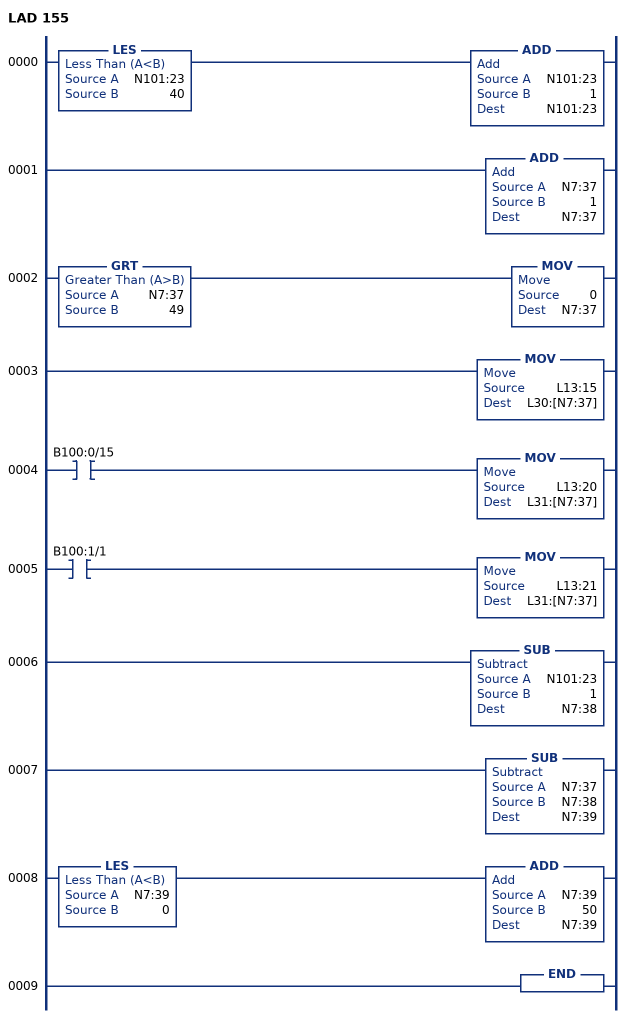
% Rung: 0 %
SOR LES N101:23 40 ADD N101:23 1 N101:23 EOR
% Rung: 1 %
SOR ADD N7:37 1 N7:37 EOR
% Rung: 2 %
SOR GRT N7:37 49 MOV 0 N7:37 EOR
% Rung: 3 %
SOR MOV L13:15 L30:[N7:37] EOR
% Rung: 4 %
SOR XIC B100:0/15 MOV L13:20 L31:[N7:37] EOR
% Rung: 5 %
SOR XIC B100:1/1 MOV L13:21 L31:[N7:37] EOR
% Rung: 6 %
SOR SUB N101:23 1 N7:38 EOR
% Rung: 7 %
SOR SUB N7:37 N7:38 N7:39 EOR
% Rung: 8 %
SOR LES N7:39 0 ADD N7:39 50 N7:39 EOR
% Rung: 9 %
SOR END EOR

LADDER 156
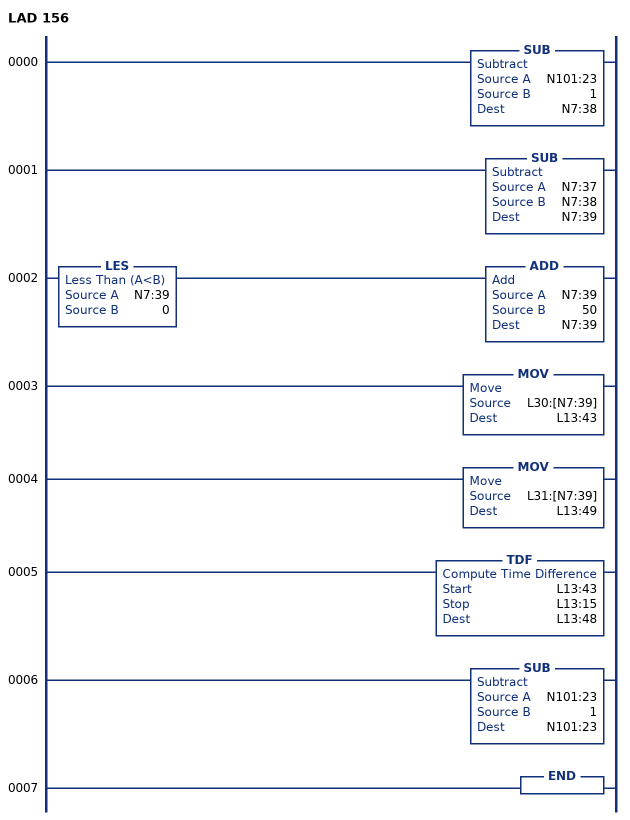
% Rung: 0 %
SOR SUB N101:23 1 N7:38 EOR
% Rung: 1 %
SOR SUB N7:37 N7:38 N7:39 EOR
% Rung: 2 %
SOR LES N7:39 0 ADD N7:39 50 N7:39 EOR
% Rung: 3 %
SOR MOV L30:[N7:39] L13:43 EOR
% Rung: 4 %
SOR MOV L31:[N7:39] L13:49 EOR
% Rung: 5 %
SOR TDF L13:43 L13:15 L13:48 EOR
% Rung: 6 %
SOR SUB N101:23 1 N101:23 EOR
% Rung: 7 %
SOR END EOR

LADDER 157
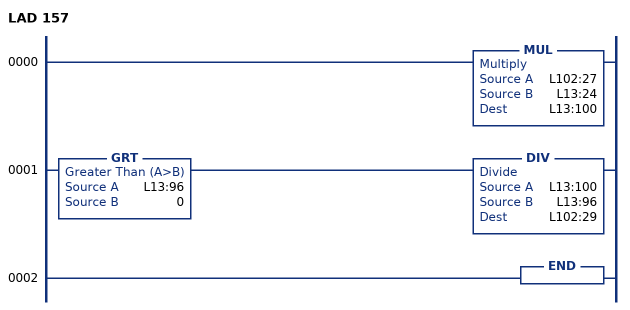
% Rung: 0 %
SOR MUL L102:27 L13:24 L13:100 EOR
% Rung: 1 %
SOR GRT L13:96 0 DIV L13:100 L13:96 L102:29 EOR
% Rung: 2 %
SOR END EOR

LADDER 158
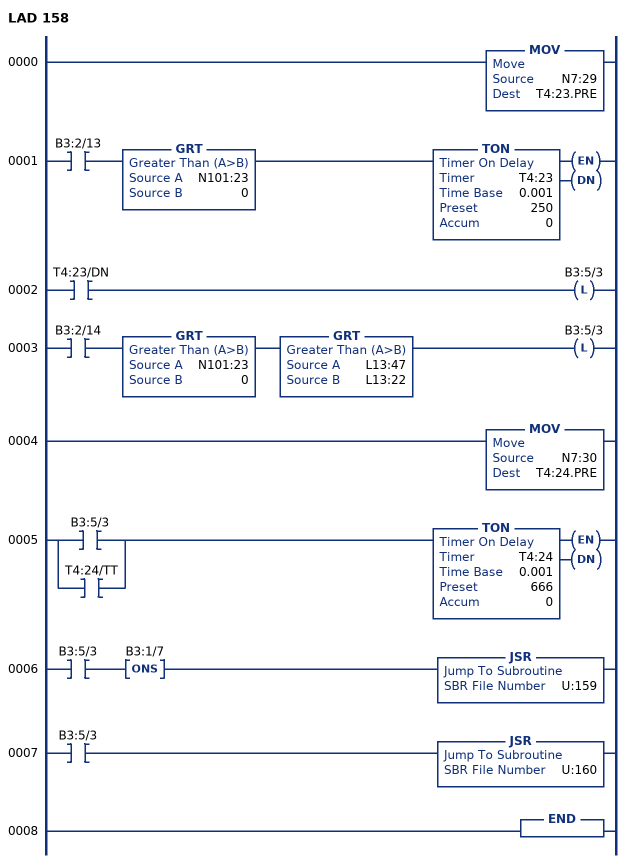
% Rung: 0 %
SOR MOV N7:29 T4:23.PRE EOR
% Rung: 1 %
SOR XIC B3:2/13 GRT N101:23 0 TON T4:23 0.001 250 0 EOR
% Rung: 2 %
SOR XIC T4:23/DN OTL B3:5/3 EOR
% Rung: 3 %
SOR XIC B3:2/14 GRT N101:23 0 GRT L13:47 L13:22 OTL B3:5/3 EOR
% Rung: 4 %
SOR MOV N7:30 T4:24.PRE EOR
% Rung: 5 %
SOR BST XIC B3:5/3 NXB XIC T4:24/TT BND TON T4:24 0.001 666 0 EOR
% Rung: 6 %
SOR XIC B3:5/3 ONS B3:1/7 JSR U:159 EOR
% Rung: 7 %
SOR XIC B3:5/3 JSR U:160 EOR
% Rung: 8 %
SOR END EOR

LADDER 159
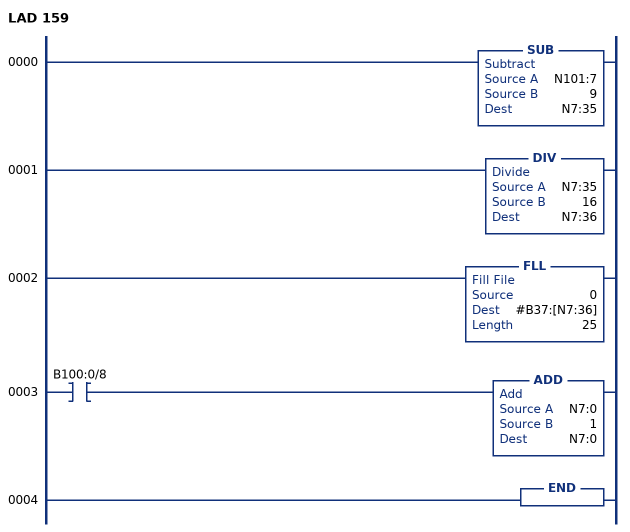
% Rung: 0 %
SOR SUB N101:7 9 N7:35 EOR
% Rung: 1 %
SOR DIV N7:35 16 N7:36 EOR
% Rung: 2 %
SOR FLL 0 #B37:[N7:36] 25 EOR
% Rung: 3 %
SOR XIC B100:0/8 ADD N7:0 1 N7:0 EOR
% Rung: 4 %
SOR END EOR

LADDER 160
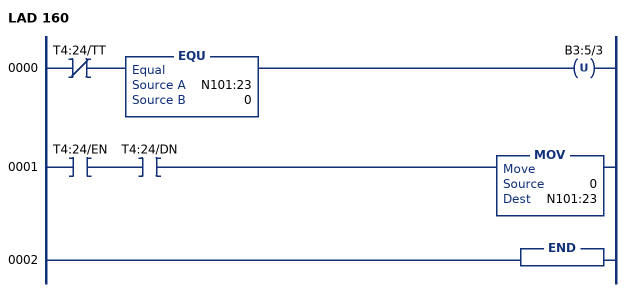
% Rung: 0 %
SOR XIO T4:24/TT EQU N101:23 0 OTU B3:5/3 EOR
% Rung: 1 %
SOR XIC T4:24/EN XIC T4:24/DN MOV 0 N101:23 EOR
% Rung: 2 %
SOR END EOR

LADDER 161
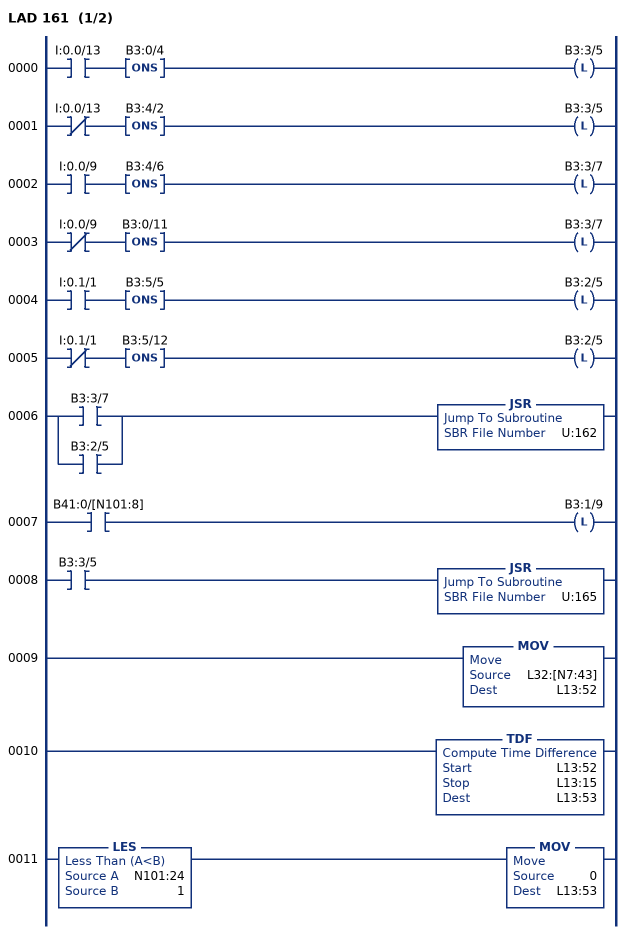
% Rung: 0 %
SOR XIC I:0.0/13 ONS B3:0/4 OTL B3:3/5 EOR
% Rung: 1 %
SOR XIO I:0.0/13 ONS B3:4/2 OTL B3:3/5 EOR
% Rung: 2 %
SOR XIC I:0.0/9 ONS B3:4/6 OTL B3:3/7 EOR
% Rung: 3 %
SOR XIO I:0.0/9 ONS B3:0/11 OTL B3:3/7 EOR
% Rung: 4 %
SOR XIC I:0.1/1 ONS B3:5/5 OTL B3:2/5 EOR
% Rung: 5 %
SOR XIO I:0.1/1 ONS B3:5/12 OTL B3:2/5 EOR
% Rung: 6 %
SOR BST XIC B3:3/7 NXB XIC B3:2/5 BND JSR U:162 EOR
% Rung: 7 %
SOR XIC B41:0/[N101:8] OTL B3:1/9 EOR
% Rung: 8 %
SOR XIC B3:3/5 JSR U:165 EOR
% Rung: 9 %
SOR MOV L32:[N7:43] L13:52 EOR
% Rung: 10 %
SOR TDF L13:52 L13:15 L13:53 EOR
% Rung: 11 %
SOR LES N101:24 1 MOV 0 L13:53 EOR

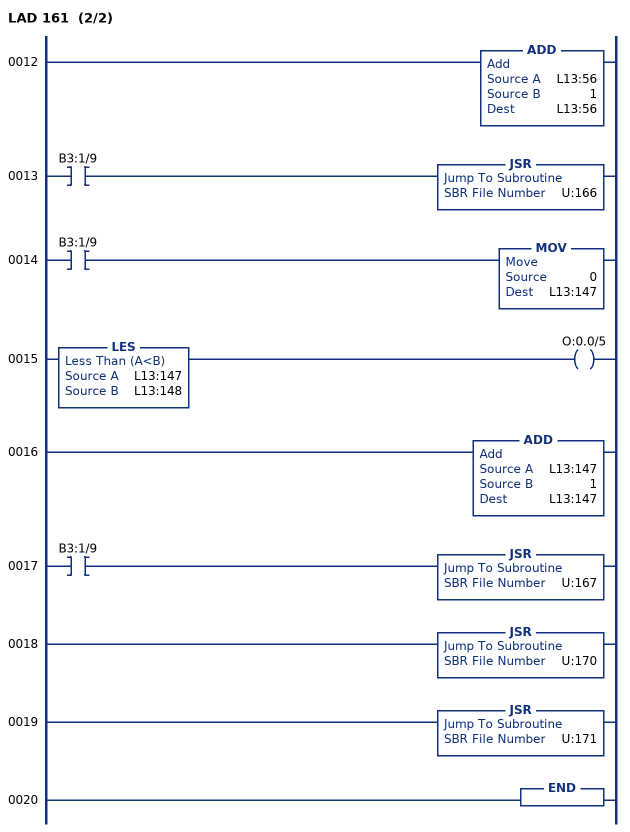
% Rung: 12 %
SOR ADD L13:56 1 L13:56 EOR
% Rung: 13 %
SOR XIC B3:1/9 JSR U:166 EOR
% Rung: 14 %
SOR XIC B3:1/9 MOV 0 L13:147 EOR
% Rung: 15 %
SOR LES L13:147 L13:148 OTE O:0.0/5 EOR
% Rung: 16 %
SOR ADD L13:147 1 L13:147 EOR
% Rung: 17 %
SOR XIC B3:1/9 JSR U:167 EOR
% Rung: 18 %
SOR JSR U:170 EOR
% Rung: 19 %
SOR JSR U:171 EOR
% Rung: 20 %
SOR END EOR

LADDER 162
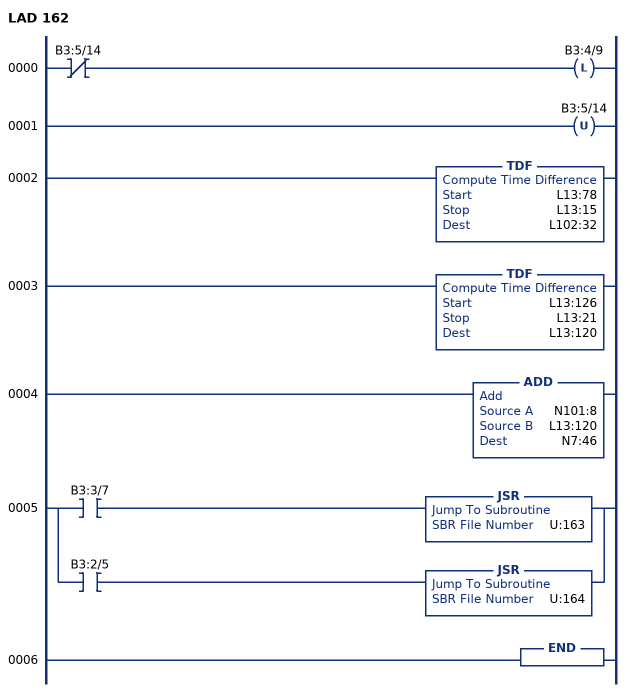
% Rung: 0 %
SOR XIO B3:5/14 OTL B3:4/9 EOR
% Rung: 1 %
SOR OTU B3:5/14 EOR
% Rung: 2 %
SOR TDF L13:78 L13:15 L102:32 EOR
% Rung: 3 %
SOR TDF L13:126 L13:21 L13:120 EOR
% Rung: 4 %
SOR ADD N101:8 L13:120 N7:46 EOR
% Rung: 5 %
SOR BST XIC B3:3/7 JSR U:163 NXB XIC B3:2/5 JSR U:164 BND EOR
% Rung: 6 %
SOR END EOR

LADDER 163
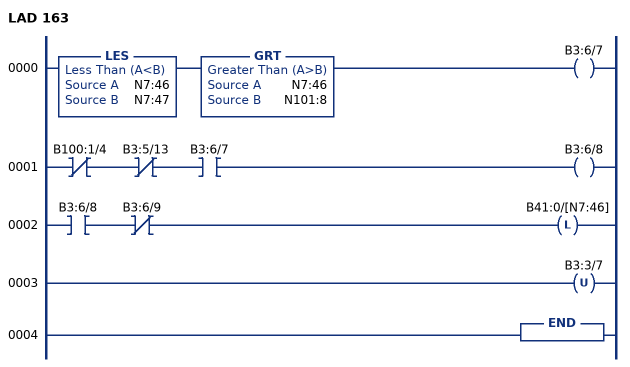
% Rung: 0 %
SOR LES N7:46 N7:47 GRT N7:46 N101:8 OTE B3:6/7 EOR
% Rung: 1 %
SOR XIO B100:1/4 XIO B3:5/13 XIC B3:6/7 OTE B3:6/8 EOR
% Rung: 2 %
SOR XIC B3:6/8 XIO B3:6/9 OTL B41:0/[N7:46] EOR
% Rung: 3 %
SOR OTU B3:3/7 EOR
% Rung: 4 %
SOR END EOR

LADDER 164
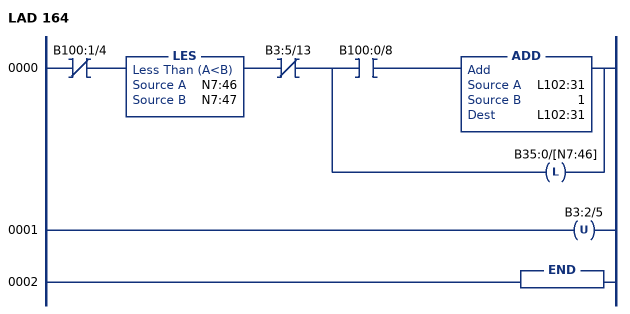
% Rung: 0 %
SOR XIO B100:1/4 LES N7:46 N7:47 XIO B3:5/13 BST XIC B100:0/8 ADD L102:31 1 L102:31 NXB OTL B35:0/[N7:46] BND EOR
% Rung: 1 %
SOR OTU B3:2/5 EOR
% Rung: 2 %
SOR END EOR

LADDER 165
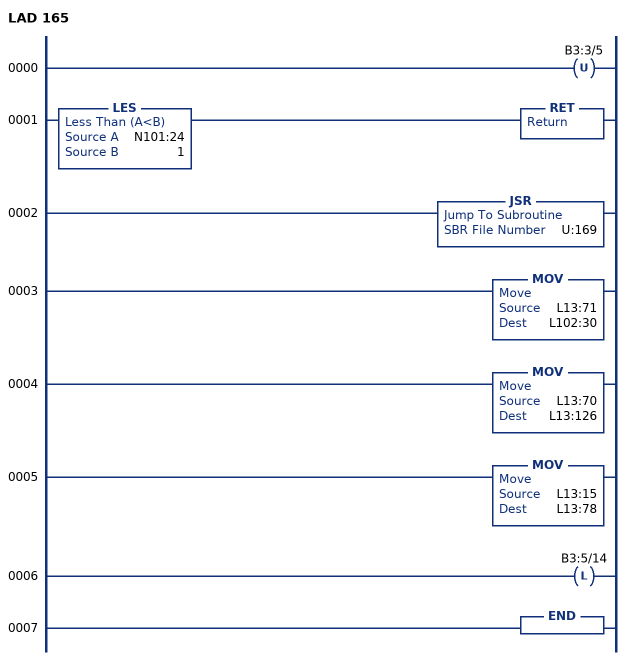
% Rung: 0 %
SOR OTU B3:3/5 EOR
% Rung: 1 %
SOR LES N101:24 1 RET EOR
% Rung: 2 %
SOR JSR U:169 EOR
% Rung: 3 %
SOR MOV L13:71 L102:30 EOR
% Rung: 4 %
SOR MOV L13:70 L13:126 EOR
% Rung: 5 %
SOR MOV L13:15 L13:78 EOR
% Rung: 6 %
SOR OTL B3:5/14 EOR
% Rung: 7 %
SOR END EOR

LADDER 166
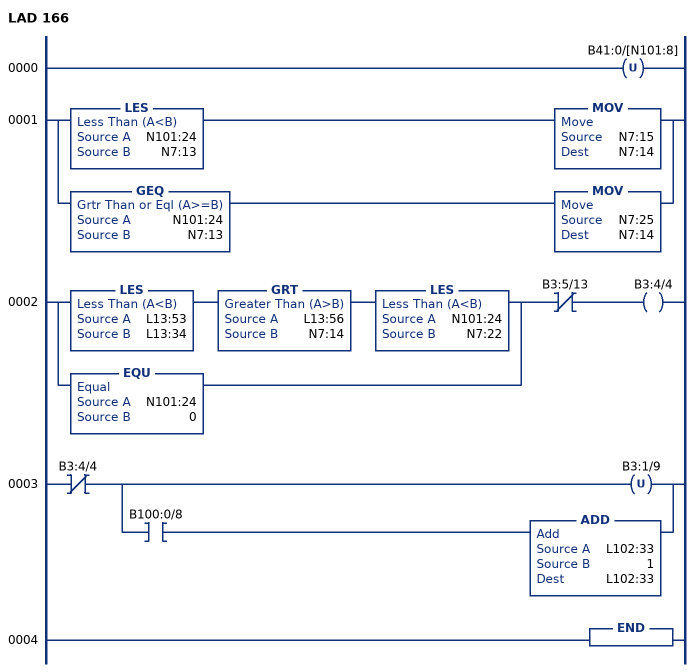
% Rung: 0 %
SOR OTU B41:0/[N101:8] EOR
% Rung: 1 %
SOR BST LES N101:24 N7:13 MOV N7:15 N7:14 NXB GEQ N101:24 N7:13 MOV N7:25 N7:14 BND EOR
% Rung: 2 %
SOR BST LES L13:53 L13:34 GRT L13:56 N7:14 LES N101:24 N7:22 NXB EQU N101:24 0 BND XIO B3:5/13 OTE B3:4/4 EOR
% Rung: 3 %
SOR XIO B3:4/4 BST OTU B3:1/9 NXB XIC B100:0/8 ADD L102:33 1 L102:33 BND EOR
% Rung: 4 %
SOR END EOR

LADDER 167
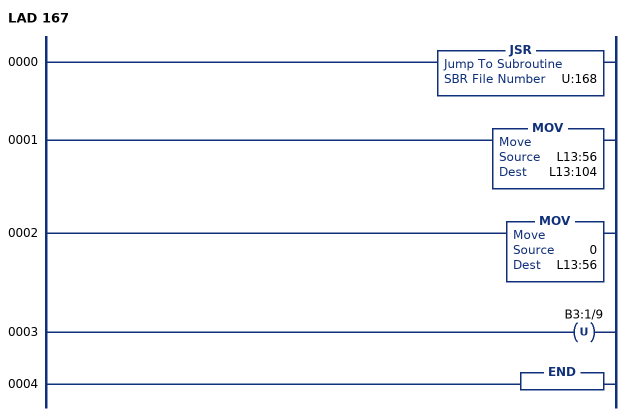
% Rung: 0 %
SOR JSR U:168 EOR
% Rung: 1 %
SOR MOV L13:56 L13:104 EOR
% Rung: 2 %
SOR MOV 0 L13:56 EOR
% Rung: 3 %
SOR OTU B3:1/9 EOR
% Rung: 4 %
SOR END EOR

LADDER 168
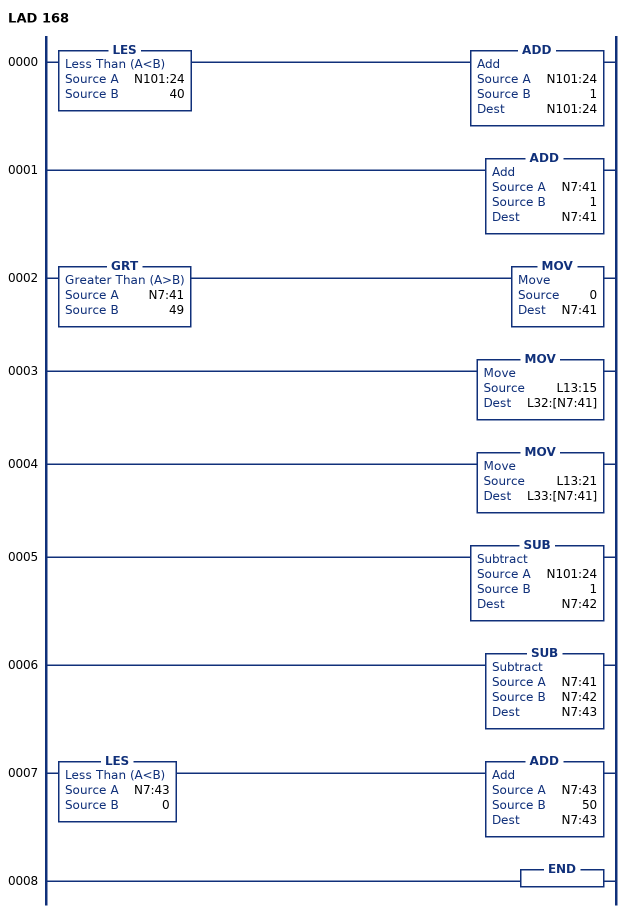
% Rung: 0 %
SOR LES N101:24 40 ADD N101:24 1 N101:24 EOR
% Rung: 1 %
SOR ADD N7:41 1 N7:41 EOR
% Rung: 2 %
SOR GRT N7:41 49 MOV 0 N7:41 EOR
% Rung: 3 %
SOR MOV L13:15 L32:[N7:41] EOR
% Rung: 4 %
SOR MOV L13:21 L33:[N7:41] EOR
% Rung: 5 %
SOR SUB N101:24 1 N7:42 EOR
% Rung: 6 %
SOR SUB N7:41 N7:42 N7:43 EOR
% Rung: 7 %
SOR LES N7:43 0 ADD N7:43 50 N7:43 EOR
% Rung: 8 %
SOR END EOR

LADDER 169
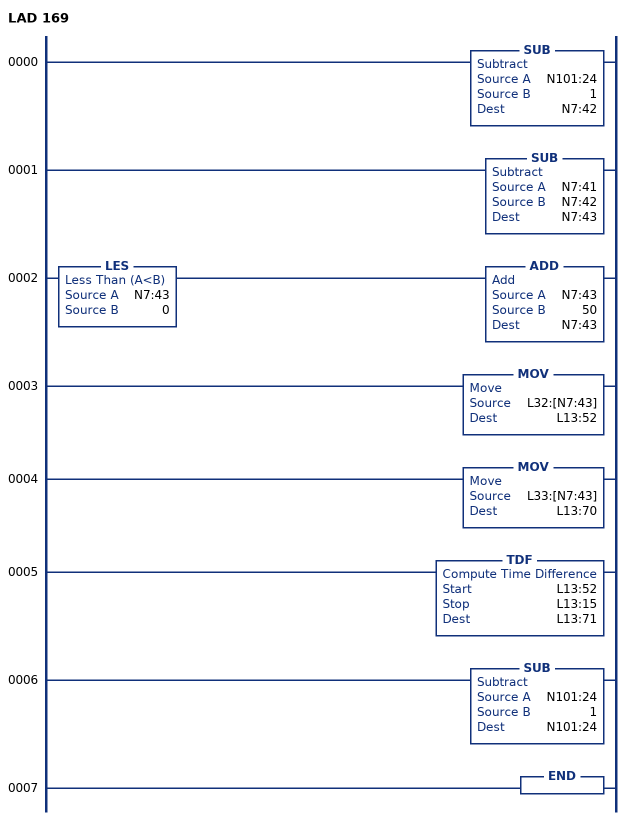
% Rung: 0 %
SOR SUB N101:24 1 N7:42 EOR
% Rung: 1 %
SOR SUB N7:41 N7:42 N7:43 EOR
% Rung: 2 %
SOR LES N7:43 0 ADD N7:43 50 N7:43 EOR
% Rung: 3 %
SOR MOV L32:[N7:43] L13:52 EOR
% Rung: 4 %
SOR MOV L33:[N7:43] L13:70 EOR
% Rung: 5 %
SOR TDF L13:52 L13:15 L13:71 EOR
% Rung: 6 %
SOR SUB N101:24 1 N101:24 EOR
% Rung: 7 %
SOR END EOR

LADDER 170
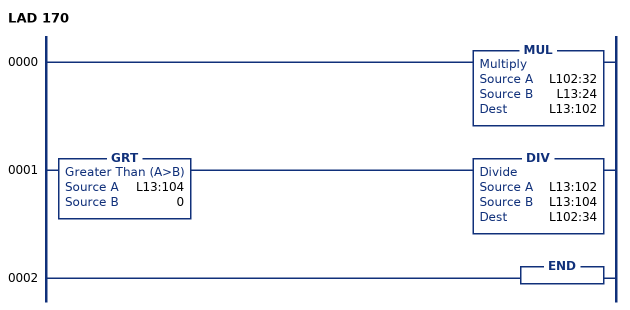
% Rung: 0 %
SOR MUL L102:32 L13:24 L13:102 EOR
% Rung: 1 %
SOR GRT L13:104 0 DIV L13:102 L13:104 L102:34 EOR
% Rung: 2 %
SOR END EOR

LADDER 171
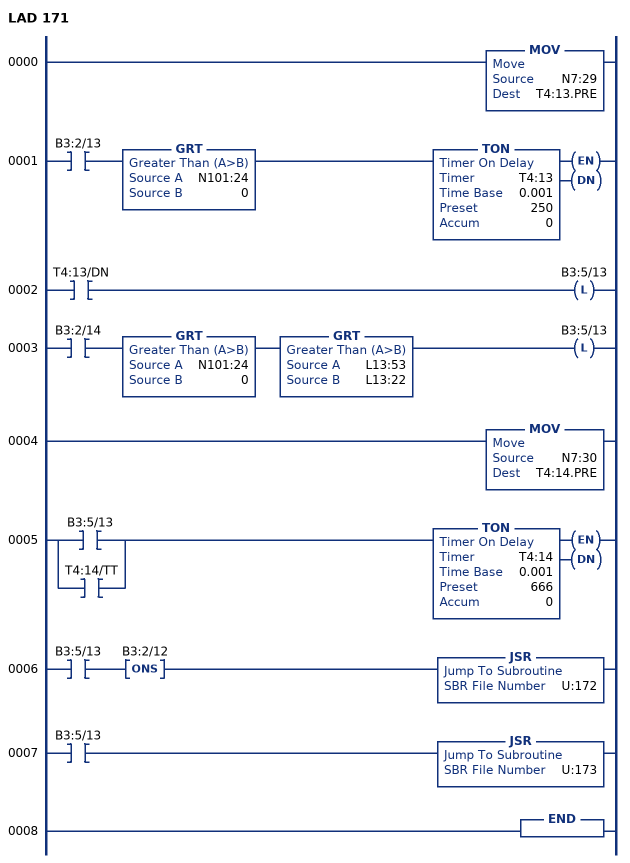
% Rung: 0 %
SOR MOV N7:29 T4:13.PRE EOR
% Rung: 1 %
SOR XIC B3:2/13 GRT N101:24 0 TON T4:13 0.001 250 0 EOR
% Rung: 2 %
SOR XIC T4:13/DN OTL B3:5/13 EOR
% Rung: 3 %
SOR XIC B3:2/14 GRT N101:24 0 GRT L13:53 L13:22 OTL B3:5/13 EOR
% Rung: 4 %
SOR MOV N7:30 T4:14.PRE EOR
% Rung: 5 %
SOR BST XIC B3:5/13 NXB XIC T4:14/TT BND TON T4:14 0.001 666 0 EOR
% Rung: 6 %
SOR XIC B3:5/13 ONS B3:2/12 JSR U:172 EOR
% Rung: 7 %
SOR XIC B3:5/13 JSR U:173 EOR
% Rung: 8 %
SOR END EOR

LADDER 172
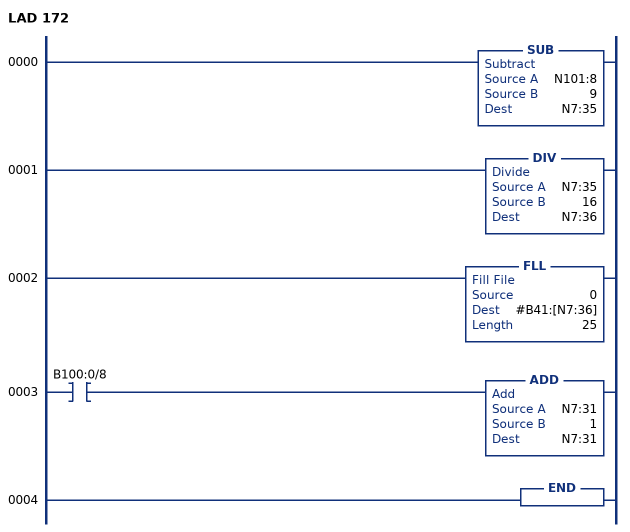
% Rung: 0 %
SOR SUB N101:8 9 N7:35 EOR
% Rung: 1 %
SOR DIV N7:35 16 N7:36 EOR
% Rung: 2 %
SOR FLL 0 #B41:[N7:36] 25 EOR
% Rung: 3 %
SOR XIC B100:0/8 ADD N7:31 1 N7:31 EOR
% Rung: 4 %
SOR END EOR

LADDER 173
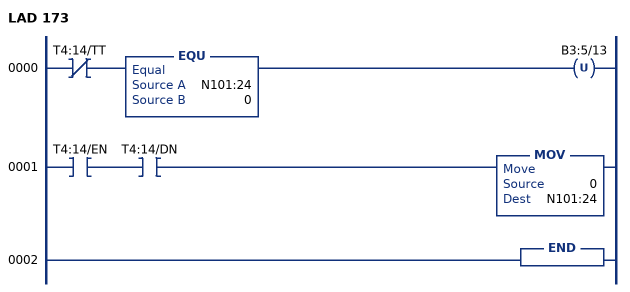
% Rung: 0 %
SOR XIO T4:14/TT EQU N101:24 0 OTU B3:5/13 EOR
% Rung: 1 %
SOR XIC T4:14/EN XIC T4:14/DN MOV 0 N101:24 EOR
% Rung: 2 %
SOR END EOR

LADDER 174
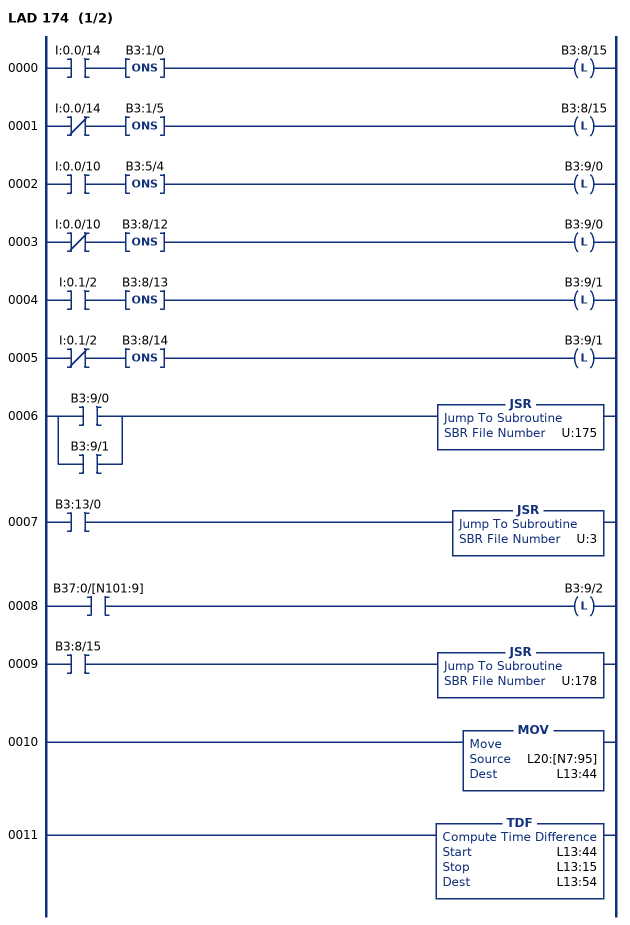
% Rung: 0 %
SOR XIC I:0.0/14 ONS B3:1/0 OTL B3:8/15 EOR
% Rung: 1 %
SOR XIO I:0.0/14 ONS B3:1/5 OTL B3:8/15 EOR
% Rung: 2 %
SOR XIC I:0.0/10 ONS B3:5/4 OTL B3:9/0 EOR
% Rung: 3 %
SOR XIO I:0.0/10 ONS B3:8/12 OTL B3:9/0 EOR
% Rung: 4 %
SOR XIC I:0.1/2 ONS B3:8/13 OTL B3:9/1 EOR
% Rung: 5 %
SOR XIO I:0.1/2 ONS B3:8/14 OTL B3:9/1 EOR
% Rung: 6 %
SOR BST XIC B3:9/0 NXB XIC B3:9/1 BND JSR U:175 EOR
% Rung: 7 %
SOR XIC B3:13/0 JSR U:3 EOR
% Rung: 8 %
SOR XIC B37:0/[N101:9] OTL B3:9/2 EOR
% Rung: 9 %
SOR XIC B3:8/15 JSR U:178 EOR
% Rung: 10 %
SOR MOV L20:[N7:95] L13:44 EOR
% Rung: 11 %
SOR TDF L13:44 L13:15 L13:54 EOR

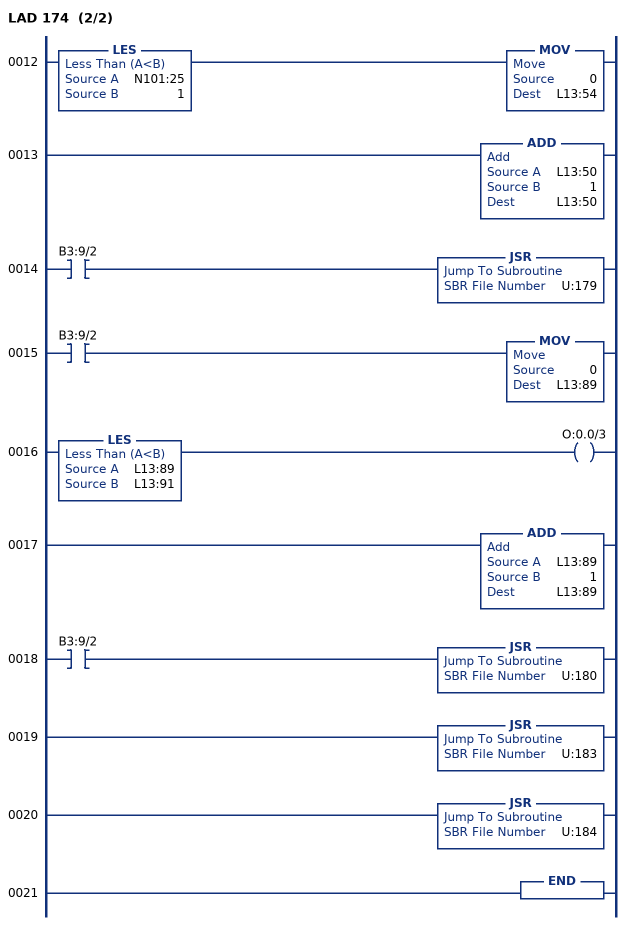
% Rung: 12 %
SOR LES N101:25 1 MOV 0 L13:54 EOR
% Rung: 13 %
SOR ADD L13:50 1 L13:50 EOR
% Rung: 14 %
SOR XIC B3:9/2 JSR U:179 EOR
% Rung: 15 %
SOR XIC B3:9/2 MOV 0 L13:89 EOR
% Rung: 16 %
SOR LES L13:89 L13:91 OTE O:0.0/3 EOR
% Rung: 17 %
SOR ADD L13:89 1 L13:89 EOR
% Rung: 18 %
SOR XIC B3:9/2 JSR U:180 EOR
% Rung: 19 %
SOR JSR U:183 EOR
% Rung: 20 %
SOR JSR U:184 EOR
% Rung: 21 %
SOR END EOR

LADDER 175
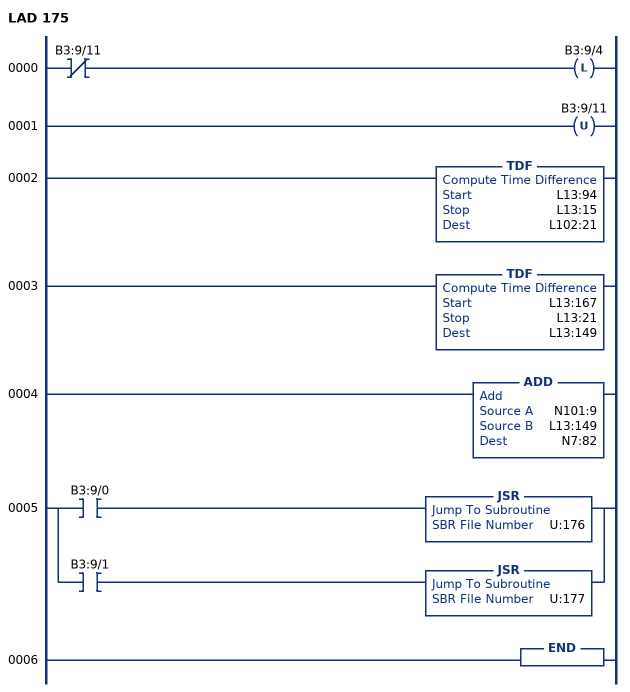
% Rung: 0 %
SOR XIO B3:9/11 OTL B3:9/4 EOR
% Rung: 1 %
SOR OTU B3:9/11 EOR
% Rung: 2 %
SOR TDF L13:94 L13:15 L102:21 EOR
% Rung: 3 %
SOR TDF L13:167 L13:21 L13:149 EOR
% Rung: 4 %
SOR ADD N101:9 L13:149 N7:82 EOR
% Rung: 5 %
SOR BST XIC B3:9/0 JSR U:176 NXB XIC B3:9/1 JSR U:177 BND EOR
% Rung: 6 %
SOR END EOR

LADDER 176
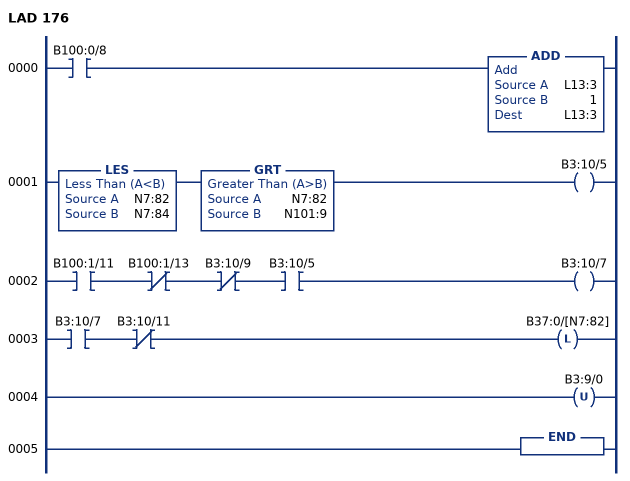
% Rung: 0 %
SOR XIC B100:0/8 ADD L13:3 1 L13:3 EOR
% Rung: 1 %
SOR LES N7:82 N7:84 GRT N7:82 N101:9 OTE B3:10/5 EOR
% Rung: 2 %
SOR XIC B100:1/11 XIO B100:1/13 XIO B3:10/9 XIC B3:10/5 OTE B3:10/7 EOR
% Rung: 3 %
SOR XIC B3:10/7 XIO B3:10/11 OTL B37:0/[N7:82] EOR
% Rung: 4 %
SOR OTU B3:9/0 EOR
% Rung: 5 %
SOR END EOR

LADDER 177
